(* IEC 61131-3 sources: Industry-PLC-LLM/data/PLCBEAD_repo/PLCBEAD_PLCEmbed-main/PLC-BEAD/Source/GEB/DATE_TO_DT, 1 file *)

(* ---- DATE_TO_DT.ST ---- *)
FUNCTION DATE_TO_DT2:UDINT
	VAR_INPUT
		IN :	UDINT;
	END_VAR
	DATE_TO_DT2 := IN;
END_FUNCTION

PROGRAM program0
  VAR
    LocalVar0 : UDINT;
	LocalOUT  : UDINT;
  END_VAR
  	LocalOUT := DATE_TO_DT2(LocalVar0);
END_PROGRAM
